TYPE PVControlMOD :
(
	PVControl_Default := 0, // 位置控制
	PVControl_Pressure := 1, // 压力控制模式
	PVControl_Other := 2 // Other
)UINT;
END_TYPE

(* stored: Version 1.1.0.1, ProductVersion 3.1.4024.4
   DUT PVControlMOD: Id {5c27c366-9b57-4e1c-baf4-814baa8d67f6} *)
